// TIA Portal V16 export
// export: Created 2021-11-12T13:31:52.7769147Z, ExportSetting WithDefaults, DisplayName Totally Integrated Automation Portal, DisplayVersion V16 Update 3, DisplayName TIA Portal Version Control Interface, DisplayVersion V16 Update 2, DisplayName TIA Portal Openness, DisplayVersion V16 Update 3, DisplayName SINAMICS Startdrive Advanced, DisplayVersion V16 Update 5, DisplayName SINAMICS Startdrive G130, G150, S120, S150, SINAMICS MV, S210, DisplayVersion V16 Update 5, DisplayName SINAMICS Startdrive G110M, G120, G120C, G120D, G120P, G115D, DisplayVersion V16 Update 5, DisplayName STEP 7 Professional, DisplayVersion V16 Update 3, DisplayName STEP 7 Safety, DisplayVersion V16, DisplayName WinCC UA Professional, DisplayVersion V16 Update 3
DATA_BLOCK "HMI_PARAM_000+UH10"   // DB59
{ S7_Optimized_Access := 'TRUE' }
VERSION : 0.1
// stored: AutoNumber true, DBAccessibleFromOPCUA true, IsOnlyStoredInLoadMemory false, IsRetainMemResEnabled false, IsWriteProtectedInAS false, MemoryReserve 100
   VAR
      xxxxx___BinarySensors___xxxxx : Byte;
      xxxxx___BinaryOthers___xxxxx : Byte;
      EC01_3 { S7_SetPoint := 'True'} : "UDT_CH_DI_Parameter";   // Chlazení rozvaděče Vstupní filtr Centrální pult UH10 OK
      FC21_14 { S7_SetPoint := 'True'} : "UDT_CH_DI_Parameter";   // Napájení 230V Centrální pult UH10 UPS OK
      FC22_14 { S7_SetPoint := 'True'} : "UDT_CH_DI_Parameter";   // Napájení 230V Centrální pult UH10 Zásuvky OK
      FB02_14 { S7_SetPoint := 'True'} : "UDT_CH_DI_Parameter";   // Napájení 230V Centrální pult UH10 Servisní zásuvky OK
      SF02_14 { S7_SetPoint := 'True'} : "UDT_CH_DI_Parameter";   // Start automat
      SF03_14 { S7_SetPoint := 'True'} : "UDT_CH_DI_Parameter";   // Nulování poruchy
      SF04_14 { S7_SetPoint := 'True'} : "UDT_CH_DI_Parameter";   // Reset bezpečnostního okruhu
      "I452.7" { S7_SetPoint := 'True'} : "UDT_CH_DI_Parameter";   // Rezerva res10
      SF06_14 { S7_SetPoint := 'True'} : "UDT_CH_DI_Parameter";   // Osvětlení kamer Zóna 1
      SF07_14 { S7_SetPoint := 'True'} : "UDT_CH_DI_Parameter";   // Osvětlení kamer Zóna 2
      SF08_14 { S7_SetPoint := 'True'} : "UDT_CH_DI_Parameter";   // Osvětlení kamer Zóna 3
      SF09_14 { S7_SetPoint := 'True'} : "UDT_CH_DI_Parameter";   // Osvětlení kamer Zóna 4
      "I453.4" { S7_SetPoint := 'True'} : "UDT_CH_DI_Parameter";   // Rezerva res15
      "I453.5" { S7_SetPoint := 'True'} : "UDT_CH_DI_Parameter";   // Rezerva res16
      "I453.7" { S7_SetPoint := 'True'} : "UDT_CH_DI_Parameter";   // Rezerva res4
      SF14_22 { S7_SetPoint := 'True'} : "UDT_CH_DI_Parameter";   // Blokování pásu v peci 1
      SF15_22 { S7_SetPoint := 'True'} : "UDT_CH_DI_Parameter";   // Blokování pásu v peci 2
      SF16_22 { S7_SetPoint := 'True'} : "UDT_CH_DI_Parameter";   // Blokování pásu v peci 3
      SF17_22 { S7_SetPoint := 'True'} : "UDT_CH_DI_Parameter";   // Blokování dopravníku chlazení 1
      SF18_22 { S7_SetPoint := 'True'} : "UDT_CH_DI_Parameter";   // Blokování pásu v peci 4
      SF19_22 { S7_SetPoint := 'True'} : "UDT_CH_DI_Parameter";   // Blokování dopravníku chlazení 2
      SF20_22 { S7_SetPoint := 'True'} : "UDT_CH_DI_Parameter";   // Blokování pásu v peci 5
      SF21_22 { S7_SetPoint := 'True'} : "UDT_CH_DI_Parameter";   // Blokování dopravníku chlazení 3
      SF22_14 { S7_SetPoint := 'True'} : "UDT_CH_DI_Parameter";   // Přemostění Safe move 2R1, 2R2
      "I455.1" { S7_SetPoint := 'True'} : "UDT_CH_DI_Parameter";   // Rezerva res14
      "I455.7" { S7_SetPoint := 'True'} : "UDT_CH_DI_Parameter";   // Rezerva res8
      "I456.1" { S7_SetPoint := 'True'} : "UDT_CH_DI_Parameter";   // Rezerva 2R3
      "I456.2" { S7_SetPoint := 'True'} : "UDT_CH_DI_Parameter";   // Rezerva 2R4
      "I456.3" { S7_SetPoint := 'True'} : "UDT_CH_DI_Parameter";   // Rezerva 2R5
      "I456.4" { S7_SetPoint := 'True'} : "UDT_CH_DI_Parameter";   // Rezerva 2R6
      "I456.5" { S7_SetPoint := 'True'} : "UDT_CH_DI_Parameter";   // Rezerva res14
      "I456.6" { S7_SetPoint := 'True'} : "UDT_CH_DI_Parameter";   // Rezerva res15
      "I456.7" { S7_SetPoint := 'True'} : "UDT_CH_DI_Parameter";   // Rezerva
      xxxxx___AnalogueSensors___xxxxx : Byte;
      xxxxx___Drives___xxxxx : Byte;
      xxxxx___Other___xxxxx : Byte;
      xxxxx___Alarms___xxxxx : Byte;
      EC01_4 { S7_SetPoint := 'True'} : "UDT_DI_Mon_Parameter";   // Chlazení rozvaděče Vstupní filtr Centrální pult UH10 OK
      FC21_15 { S7_SetPoint := 'True'} : "UDT_DI_Mon_Parameter";   // Napájení 230V Centrální pult UH10 UPS OK
      FC22_15 { S7_SetPoint := 'True'} : "UDT_DI_Mon_Parameter";   // Napájení 230V Centrální pult UH10 Zásuvky OK
      FB02_15 { S7_SetPoint := 'True'} : "UDT_DI_Mon_Parameter";   // Napájení 230V Centrální pult UH10 Servisní zásuvky OK
      SF22_15 { S7_SetPoint := 'True'} : "UDT_DI_Mon_Parameter";   // Přemostění Safe move 2R1, 2R2
      ES { S7_SetPoint := 'True'} : "UDT_DI_Mon_Parameter";   // E-stop
   END_VAR
BEGIN
END_DATA_BLOCK
